INTERFACE I_EnumeratorConnection

METHOD PUBLIC SetInvalid
VAR_INPUT
END_VAR
END_METHOD

END_INTERFACE

(* stored: Version 1.1.0.1, ProductVersion 3.1.4024.12
   Itf I_EnumeratorConnection: Id {8f9feb07-0a4c-4839-9083-e25e6864c9fc}
   Method SetInvalid: Id {68b4f5b5-ca02-4533-b0f0-393b978fc52b} *)
